FUNCTION_BLOCK FlexPRET
  (* Standard: 61499-2 *)
  (* Version 0.1, 2016-00-28, hpea485, UOA *)
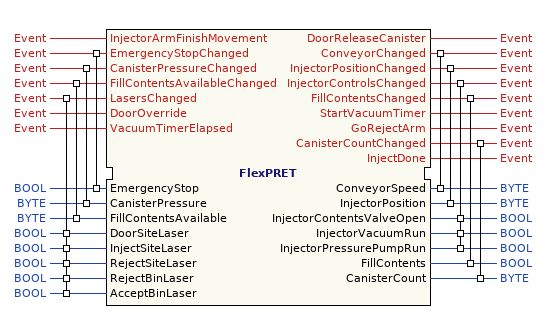
  EVENT_INPUT
    InjectorArmFinishMovement;
    EmergencyStopChanged WITH EmergencyStop;
    CanisterPressureChanged WITH CanisterPressure;
    FillContentsAvailableChanged WITH FillContentsAvailable;
    LasersChanged WITH DoorSiteLaser, InjectSiteLaser, RejectSiteLaser, RejectBinLaser, AcceptBinLaser;
    DoorOverride;
    VacuumTimerElapsed;
  END_EVENT
  EVENT_OUTPUT
    DoorReleaseCanister;
    ConveyorChanged WITH ConveyorSpeed;
    InjectorPositionChanged WITH InjectorPosition;
    InjectorControlsChanged WITH InjectorContentsValveOpen, InjectorVacuumRun, InjectorPressurePumpRun;
    FillContentsChanged WITH FillContents;
    StartVacuumTimer;
    GoRejectArm;
    CanisterCountChanged WITH CanisterCount;
    InjectDone;
  END_EVENT
  VAR_INPUT
    EmergencyStop : BOOL;
    CanisterPressure : BYTE;
    FillContentsAvailable : BYTE;
    DoorSiteLaser : BOOL;
    InjectSiteLaser : BOOL;
    RejectSiteLaser : BOOL;
    RejectBinLaser : BOOL;
    AcceptBinLaser : BOOL;
  END_VAR
  VAR_OUTPUT
    ConveyorSpeed : BYTE;
    InjectorPosition : BYTE;
    InjectorContentsValveOpen : BOOL;
    InjectorVacuumRun : BOOL;
    InjectorPressurePumpRun : BOOL;
    FillContents : BOOL;
    CanisterCount : BYTE;
  END_VAR
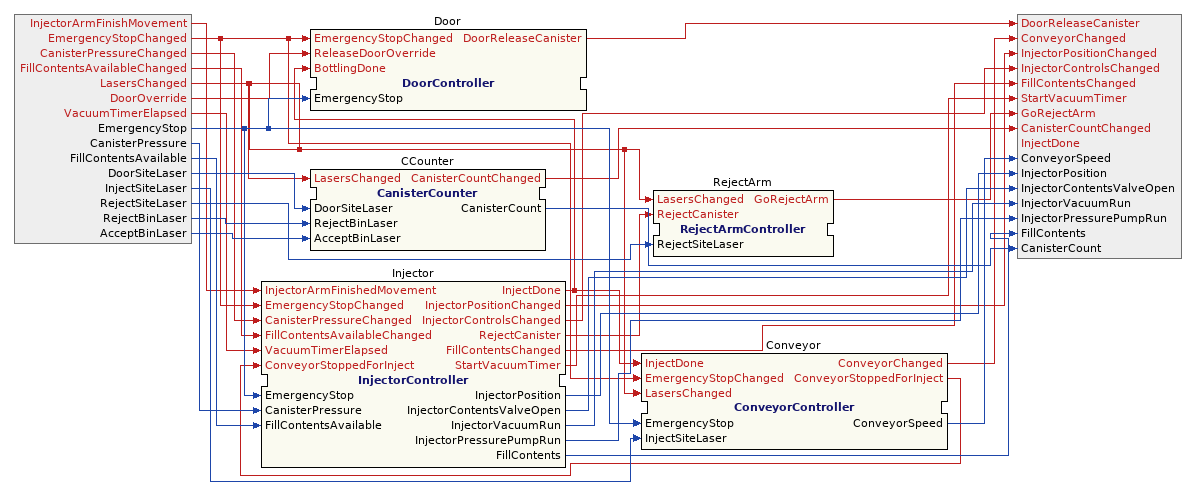
  FBS
    CCounter : CanisterCounter;
    Door : DoorController;
    Injector : InjectorController;
    Conveyor : ConveyorController;
    RejectArm : RejectArmController;
  END_FBS
  EVENT_CONNECTIONS
    InjectorArmFinishMovement TO Injector.InjectorArmFinishedMovement;
    EmergencyStopChanged TO Door.EmergencyStopChanged;
    EmergencyStopChanged TO Injector.EmergencyStopChanged;
    EmergencyStopChanged TO Conveyor.EmergencyStopChanged;
    CanisterPressureChanged TO Injector.CanisterPressureChanged;
    FillContentsAvailableChanged TO Injector.FillContentsAvailableChanged;
    LasersChanged TO CCounter.LasersChanged;
    LasersChanged TO RejectArm.LasersChanged;
    LasersChanged TO Conveyor.LasersChanged;
    DoorOverride TO Door.ReleaseDoorOverride;
    VacuumTimerElapsed TO Injector.VacuumTimerElapsed;
    CCounter.CanisterCountChanged TO CanisterCountChanged;
    Door.DoorReleaseCanister TO DoorReleaseCanister;
    Injector.InjectDone TO Door.BottlingDone;
    Injector.InjectDone TO Conveyor.InjectDone;
    Injector.InjectorPositionChanged TO InjectorPositionChanged;
    Injector.InjectorControlsChanged TO InjectorControlsChanged;
    Injector.RejectCanister TO RejectArm.RejectCanister;
    Injector.FillContentsChanged TO FillContentsChanged;
    Injector.StartVacuumTimer TO StartVacuumTimer;
    Conveyor.ConveyorChanged TO ConveyorChanged;
    Conveyor.ConveyorStoppedForInject TO Injector.ConveyorStoppedForInject;
    RejectArm.GoRejectArm TO GoRejectArm;
  END_CONNECTIONS
  DATA_CONNECTIONS
    EmergencyStop TO Door.EmergencyStop;
    EmergencyStop TO Injector.EmergencyStop;
    EmergencyStop TO Conveyor.EmergencyStop;
    CanisterPressure TO Injector.CanisterPressure;
    FillContentsAvailable TO Injector.FillContentsAvailable;
    DoorSiteLaser TO CCounter.DoorSiteLaser;
    InjectSiteLaser TO Conveyor.InjectSiteLaser;
    RejectSiteLaser TO RejectArm.RejectSiteLaser;
    RejectBinLaser TO CCounter.RejectBinLaser;
    AcceptBinLaser TO CCounter.AcceptBinLaser;
    CCounter.CanisterCount TO CanisterCount;
    Injector.InjectorPosition TO InjectorPosition;
    Injector.InjectorContentsValveOpen TO InjectorContentsValveOpen;
    Injector.InjectorVacuumRun TO InjectorVacuumRun;
    Injector.InjectorPressurePumpRun TO InjectorPressurePumpRun;
    Injector.FillContents TO FillContents;
    Conveyor.ConveyorSpeed TO ConveyorSpeed;
  END_CONNECTIONS
END_FUNCTION_BLOCK
